FUNCTION TFPalletizer_CalcolaCoordinataPrelievo_PickPoint : LREAL
VAR_INPUT
	WorkPickPoint : POINTER TO ARRAY [1..MAXPICKPOINT] OF TFMachinePalletizer_WorkPickPointSlab;
	WorkPickPointState : POINTER TO ARRAY [1..MAXPICKPOINT] OF TFMachinePalletizer_WorkPickPoint_State;
	WorkPickPointOffset : POINTER TO ARRAY [1..MAXPICKPOINT] OF TFMachinePalletizer_WorkPickPointOffset;
	NPickPoint : UINT;			//Numero PickPoint del quale si vuole la coordinata
	AsseDaCalcolare : STRING;	//Nome dell'Asse del quale si vuole calcolare la coordinata 
END_VAR
VAR
	wpp : INT;
	Ncase : INT;
END_VAR

TFPalletizer_CalcolaCoordinataPrelievo_PickPoint := 0;
IF AsseDaCalcolare = 'X' THEN
	Ncase	:= 1;
ELSIF AsseDaCalcolare = 'Y' THEN
	Ncase	:= 2;
ELSIF AsseDaCalcolare = 'Z' THEN
	Ncase	:= 3;
ELSIF AsseDaCalcolare = 'J' THEN
	Ncase	:= 4;
END_IF

IF WorkPickPoint^[NPickPoint].Tipologia = WA_CON_PALLET  OR WorkPickPoint^[NPickPoint].Tipologia = WA_CON_CASSA OR WorkPickPoint^[NPickPoint].Tipologia = WA_CON_CAVALLINA THEN
	CASE Ncase OF
		1:
			TFPalletizer_CalcolaCoordinataPrelievo_PickPoint := WorkPickPoint^[NPickPoint].X +							// Quota X centro Rulliera	
																//WorkPickPointState^[NPickPoint].XPosBandella +	// Quota Relativa della posizione della bandella
																//(WorkPickPointState^[NPickPoint].Element.XDim/2) +		// Metà Lunghezza Lastra
																WorkPickPointOffset^[NPickPoint].X;						// Valore di Offset Di Prelievo in X	
		
		2:	
			TFPalletizer_CalcolaCoordinataPrelievo_PickPoint := WorkPickPoint^[NPickPoint].Y -							// Quota Y centro Rulliera	
																//WorkPickPointState^[NPickPoint].YPosBandella +	// Quota Relativa della posizione della bandella
																(WorkPickPointState^[NPickPoint].Element.YDim/2) +		// Metà Larghezza Lastra
																WorkPickPointOffset^[NPickPoint].Y;						// Valore di Offset Di Prelievo in Y
		3:	
			TFPalletizer_CalcolaCoordinataPrelievo_PickPoint := WorkPickPoint^[NPickPoint].Z +							// Quota Z, altezza della postazione
																WorkPickPointState^[NPickPoint].Element.ZDim +			// Metà Larghezza Lastra
																WorkPickPointOffset^[NPickPoint].Z;						// Valore di Offset Di Prelievo in Y
		4:	
			TFPalletizer_CalcolaCoordinataPrelievo_PickPoint := WorkPickPoint^[NPickPoint].J +							// Quota Y centro Rulliera	
																WorkPickPointOffset^[NPickPoint].J;						// Valore di Offset Di Prelievo in Y	
	END_CASE
ELSE
	CASE Ncase OF
		1:
			//TFPalletizer_CalcolaCoordinataPrelievo_PickPoint := WorkPickPoint^[NPickPoint].X +							// Quota X centro Rulliera	
			//													//WorkPickPointState^[NPickPoint].XPosBandella +	// Quota Relativa della posizione della bandella
			//													//(WorkPickPointState^[NPickPoint].Element.XDim/2) +		// Metà Lunghezza Lastra
			//													WorkPickPointOffset^[NPickPoint].X;						// Valore di Offset Di Prelievo in X	
		
			CASE TIPOLOGIA_RULLIERA_PRELIEVO OF
					
				RULLIERA_LONGITUDINALE:
										TFPalletizer_CalcolaCoordinataPrelievo_PickPoint := WorkPickPoint^[NPickPoint].X -							// Quota X centro Rulliera	
																//WorkPickPointState^[NPickPoint].XPosBandella +	// Quota Relativa della posizione della bandella
																//(WorkPickPointState^[NPickPoint].Element.XDim/2) +		// Metà Lunghezza Lastra
																MAX(Dimensioni_Pinza.Lunghezza/2,WorkPickPointState^[NPickPoint].Element.XDim/2) +
																WorkPickPointOffset^[NPickPoint].X;						// Valore di Offset Di Prelievo in X	
		
					
				RULLIERA_TRASVERSALE:
										TFPalletizer_CalcolaCoordinataPrelievo_PickPoint := WorkPickPoint^[NPickPoint].X +							// Quota X centro Rulliera	
																//WorkPickPointState^[NPickPoint].XPosBandella +	// Quota Relativa della posizione della bandella
																//(WorkPickPointState^[NPickPoint].Element.XDim/2) +		// Metà Lunghezza Lastra
																WorkPickPointOffset^[NPickPoint].X;						// Valore di Offset Di Prelievo in X	
									
			END_CASE
													
		2:	
			//TFPalletizer_CalcolaCoordinataPrelievo_PickPoint := WorkPickPoint^[NPickPoint].Y -							// Quota Y centro Rulliera	
			//												//	WorkPickPointState^[NPickPoint].YPosBandella +	// Quota Relativa della posizione della bandella
			//													(WorkPickPointState^[NPickPoint].Element.YDim/2) +		// Metà Larghezza Lastra
			//													WorkPickPointOffset^[NPickPoint].Y;						// Valore di Offset Di Prelievo in Y
	
			CASE TIPOLOGIA_RULLIERA_PRELIEVO OF
					
				RULLIERA_LONGITUDINALE:
										TFPalletizer_CalcolaCoordinataPrelievo_PickPoint := WorkPickPoint^[NPickPoint].Y +							// Quota Y centro Rulliera	
															//	WorkPickPointState^[NPickPoint].YPosBandella +	// Quota Relativa della posizione della bandella
															//	(WorkPickPointState^[NPickPoint].Element.YDim/2) +		// Metà Larghezza Lastra
																WorkPickPointOffset^[NPickPoint].Y;						// Valore di Offset Di Prelievo in Y
				RULLIERA_TRASVERSALE:
										TFPalletizer_CalcolaCoordinataPrelievo_PickPoint := WorkPickPoint^[NPickPoint].Y -							// Quota Y centro Rulliera	
															//	WorkPickPointState^[NPickPoint].YPosBandella +	// Quota Relativa della posizione della bandella
																(WorkPickPointState^[NPickPoint].Element.YDim/2) +		// Metà Larghezza Lastra
																WorkPickPointOffset^[NPickPoint].Y;						// Valore di Offset Di Prelievo in Y
				
			END_CASE


		3:	
			TFPalletizer_CalcolaCoordinataPrelievo_PickPoint := WorkPickPoint^[NPickPoint].Z +							// Quota Y centro Rulliera	
																WorkPickPointState^[NPickPoint].Element.ZDim +			// Metà Larghezza Lastra
																WorkPickPointOffset^[NPickPoint].Z;						// Valore di Offset Di Prelievo in Y
		4:	
			TFPalletizer_CalcolaCoordinataPrelievo_PickPoint := WorkPickPoint^[NPickPoint].J +							// Quota Y centro Rulliera	
																WorkPickPointOffset^[NPickPoint].J;						// Valore di Offset Di Prelievo in Y	
	END_CASE
END_IF

END_FUNCTION

(* stored: Version 1.1.0.1, ProductVersion 3.1.4024.11
   POU TFPalletizer_CalcolaCoordinataPrelievo_PickPoint: Id {916aecfa-a0c5-4a42-9262-1c9ca786d9ac}, SpecialFunc None *)
